FUNCTION_BLOCK FB_HYST_3 (* Basic Function Block Type *)
  (* Standard: 61499-2 *)
  (* Version 0.0, 2011-08-31, 4DIAC-IDE, 4DIAC-Consortium *)
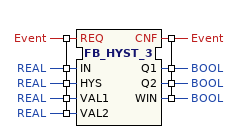
  EVENT_INPUT
    REQ WITH IN, VAL1, HYS, VAL2; (* Normal Execution Request *)
  END_EVENT
  EVENT_OUTPUT
    CNF WITH WIN, Q1, Q2; (* Execution Confirmation *)
  END_EVENT
  VAR_INPUT
    IN : REAL; (* input value *)
    HYS : REAL; (* width of the hysteresis *)
    VAL1 : REAL; (* mean of the hysteresis 1 *)
    VAL2 : REAL; (* mean of hysteresis 2 *)
  END_VAR
  VAR_OUTPUT
    Q1 : BOOL; (* output *)
    Q2 : BOOL; (* output 2 *)
    WIN : BOOL; (* shows that IN lies in the window *)
  END_VAR
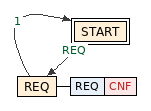
  EC_STATES
    START; (* Initial State *)
    REQ : REQ -> CNF; (* Normal execution *)
  END_STATES
  EC_TRANSITIONS
    START TO REQ := REQ;
    REQ TO START := 1;
  END_TRANSITIONS
  ALGORITHM REQ IN ST: (* Normally executed algorithm *)
VAR
	X: REAL;
END_VAR

X := HYS * 0.5;

IF IN < VAL1 - X THEN
	Q1 := TRUE;
ELSIF IN > VAL1 + X THEN
	Q1 := FALSE;
END_IF;

IF IN < VAL2 - X THEN
	Q2 := FALSE;
ELSIF IN > VAL2 + X THEN
	Q2 := TRUE;
END_IF;
  END_ALGORITHM
END_FUNCTION_BLOCK
